(* PLC project PRG_GLOBAL_CFC.project, Dragage CODESYS CODESYS V3.5 SP19 Patch 1 *)
(* stored: creationDateTime 2026-07-30T01:21:00, modificationDateTime 2026-07-30T01:21:00 *)

PROGRAM PRG_GLOBAL_CFC
  VAR
    instDiagCanOpen : FB_DiagCanOpen;
    instModes : FB_Modes;
    instCycle : FB_Cycle;
  END_VAR

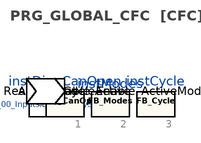
(* CFC diagram, written out as Structured Text *)
instDiagCanOpen(Enable := PRG_00_Inputs.EmergencyStopOk);
instModes(Enable := instDiagCanOpen.Ready);
instCycle(ActiveMode := instModes.ActiveMode);
END_PROGRAM
